(* Logix 5000 project; controller Contador Emulate 5570 rev 30.12; software revision 30.00 *)

TASK MainTask (continuous, watchdog 500 ms) : MainProgram

MODULES
   Local : Emulate 5570 (ICP 2, rev 30.12)
      I_O : vendor 1 type 0 code 15 (ICP 3, rev 1.1, Output RPI 150 ms)
END_MODULES

VAR_GLOBAL   (* controller tags *)
   Activar : BOOL;
   Banda1 : BOOL;
   Banda2 : BOOL;
   BanderaS2 : BOOL := 1;
   Barra : BOOL;
   FB_sensor2 : BOOL;
   Parada : BOOL;
   Sensor2 : BOOL := 1;
   Sensor3 : BOOL := 1;
   Start : BOOL;
   Stop : BOOL := 1;
   Stop_emergencia : BOOL := 1;
   TimerBa : TIMER := (PRE := 2000, ACC := 2000);
   TimerBaUp : TIMER := (PRE := 1700);
   TimerS3 : TIMER := (PRE := 4000);
END_VAR

PROGRAM MainProgram   (* main routine MainRoutine *)
VAR
   Counter1 : COUNTER := (PRE := 5);
END_VAR

ROUTINE MainRoutine   (* ladder *)
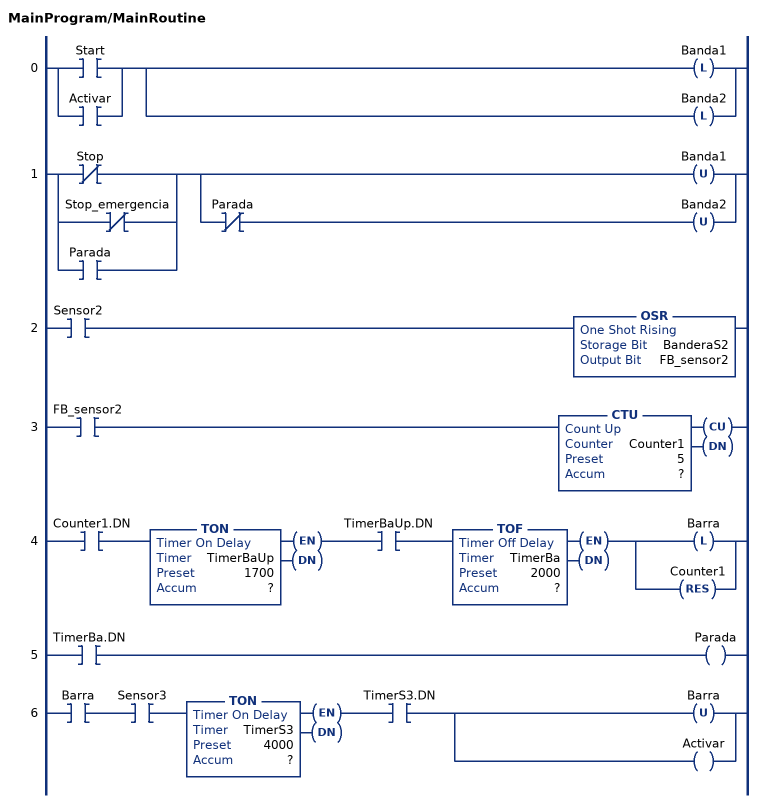
   0: [XIC(Start) ,XIC(Activar) ][OTL(Banda1) ,OTL(Banda2) ];
   1: [XIO(Stop) ,XIO(Stop_emergencia) ,XIC(Parada) ][OTU(Banda1) ,XIO(Parada) OTU(Banda2) ];
   2: XIC(Sensor2)OSR(BanderaS2,FB_sensor2);
   3: XIC(FB_sensor2)CTU(Counter1,?,?);
   4: XIC(Counter1.DN)TON(TimerBaUp,?,?)XIC(TimerBaUp.DN)TOF(TimerBa,?,?)[OTL(Barra) ,RES(Counter1) ];
   5: XIC(TimerBa.DN)OTE(Parada);
   6: XIC(Barra)XIC(Sensor3)TON(TimerS3,?,?)XIC(TimerS3.DN)[OTU(Barra) ,OTE(Activar) ];
END_ROUTINE
END_PROGRAM
